Cover2_error := Cover2_opened AND Cover2_closed;
Cover3_error := Cover3_opened AND Cover3_closed;
// we are open, if all covers are open
isopen := cover3_opened AND cover2_opened;
// we are closed, if all covers are closed
isclosed := cover2_closed AND cover3_closed;
// error indicates an axis error on any axis
Cover2_timeout(IN := (open AND NOT Cover2_opened) OR (close AND NOT Cover2_closed), PT := T#30S);
Cover3_timeout(IN := (open AND NOT Cover3_opened) OR (close AND NOT Cover3_closed), PT := T#30S);

error_trigger(	SET1 := Cover2_error OR Cover2_timeout.Q OR Cover3_error OR Cover3_timeout.Q,
				RESET := reset,
				Q1 => Error);

Ready := NOT Error;

IF isopen THEN
	open := FALSE;
END_IF
IF isclosed THEN
	close := FALSE;
END_IF

Cover_status.0 := isopen;
Cover_status.1 := isclosed;
Cover_status.2 := Warning;
Cover_status.3 := Error;
Cover_status.4 := isopen;
Cover_status.5 := FALSE;
Cover_status.6 := Cover2_opened;
Cover_status.7 := Cover3_opened;
Cover_status.8 := FALSE;
Cover_status.9 := Cover2_closed;
Cover_status.10 := Cover3_closed;
Cover_status.11 := FALSE;
Cover_status.12 := Cover2_error;
Cover_status.13 := Cover3_error;

IF Cover_status <> LastStatus THEN
	LastStatus := Cover_status;
	MAIN.MQTTClient.Publish('telescope', 'cover', 'CoverIsOpen', BOOL_TO_STRING(isopen));
	MAIN.MQTTClient.Publish('telescope', 'cover', 'CoverIsClosed', BOOL_TO_STRING(isclosed));
	MAIN.MQTTClient.Publish('telescope', 'cover', 'CoverWarning', BOOL_TO_STRING(Warning));
	MAIN.MQTTClient.Publish('telescope', 'cover', 'CoverError', BOOL_TO_STRING(Error));
	MAIN.MQTTClient.Publish('telescope', 'cover', 'CoverStatus', WORD_TO_STRING(Cover_status));
END_IF

// A timeout occurs, when we open the cover, and the opened signal does not activate within n seconds.
// The same holds for closing the cover. This should not take longer then 10 seconds
Cover2_timeout(IN := NOT (Cover2_opened XOR Cover2_closed), PT := T#20S);
				
Cover3_timeout(IN := NOT (Cover3_opened XOR Cover3_closed), PT := T#20S);

Covers_Error_Event.OnMessage := 'Cover drive error';
IF Error THEN
	IF Cover3_error THEN 
		Covers_Error_Event.OnMessage := 'Cover 3 has a drive error.';
	END_IF
	IF Cover2_error THEN 
		Covers_Error_Event.OnMessage := 'Cover 2 has a drive error.';
	END_IF
END_IF


Covers_Error_event(	Trigger := Error, 
					Level := ADSLOG_MSGTYPE_ERROR);

Covers_Warning_event(	Trigger := Warning, 
						Level := ADSLOG_MSGTYPE_WARN);

// raise an error, if both opened and closed signals are activated
// handle RoboTel differently
Cover2_Event(Trigger := cover2_opened AND cover2_closed,
				Level := ADSLOG_MSGTYPE_ERROR, 
				OnMessage := 'Cover2: limit switch error');

Cover3_Event(Trigger := cover3_opened AND cover3_closed,
				Level := ADSLOG_MSGTYPE_ERROR, 
				OnMessage := 'Cover3: limit switch error');

//trigger an event, if we encounter a timeout
// handle RoboTel differently

Cover2_Timeout_Event(Trigger := Cover2_timeout.Q,
				Level := ADSLOG_MSGTYPE_ERROR, 
				OnMessage := 'Cover2: Timeout');

Cover3_Timeout_Event(Trigger := Cover3_timeout.Q,
				Level := ADSLOG_MSGTYPE_ERROR, 
				OnMessage := 'Cover3: Timeout');
// Log if we are opened
Covers_opened_event(Trigger := isopen,
					Level := ADSLOG_MSGTYPE_WARN,
					OnMessage := 'All covers are open');
//log if we are closed
Covers_closed_event(Trigger := isclosed,
					Level := ADSLOG_MSGTYPE_HINT,
					OnMessage := 'All covers are closed');

END_PROGRAM

// ---- POUs/NasmythControl.TcPOU
PROGRAM NasmythControl
VAR_INPUT
	// unlocks the brake and enables the drive
	enable:	BOOL;
	// resets the drive
	reset: BOOL;
	// turns the Nasmyth mirror to left port (seen from top)
	left:	BOOL;
	// turns the Nasmyth mirror to right port (seen from top)
	right:	BOOL;
END_VAR
VAR_OUTPUT
	// Nasmyth drive error
	error:	BOOL;
	// drive ready
	Ready:	BOOL;
	// Nasmyth points to right mirror
	Nasmyth_right:		BOOL;
	// Nasmyth points to left mirror
	Nasmyth_left:		BOOL;
END_VAR
VAR
	//move to derotator
	nasmyth_move_left	AT%Q*: BOOL;
	nasmyth_move_right	AT%Q*: BOOL;
	// delay for the Nasmyth holding brake
	Nasmyth_delay:		TON;
	// status word for MQTT message
	Nasmyth_status:		WORD;
	// last status word to trigger MQTT message if different
	LastStatus:			WORD;
	// unlock the holding brake
	Nasmyth_unlock:		BOOL;
	// holding brake is unlocked
	Nasmyth_unlocked:	BOOL;
	// event log of error
	NasmythEvent: 		FB_Eventlog;
	NasmythLeftEvent:	FB_Eventlog;
	NasmythRightEvent:	FB_Eventlog;
	Nasmyth_Timeout:	TON := (PT := T#10S);
END_VAR

// get the inputs
Nasmyth_left := GVL_Telescope.nasmyth_limit_right;
Nasmyth_right := GVL_Telescope.nasmyth_limit_left;

// disable command, if position has been reached or 
IF Nasmyth_left OR right THEN
	left := FALSE;
END_IF

IF  Nasmyth_right OR left THEN
	right := FALSE;
END_IF

Nasmyth_status.0 := Nasmyth_unlocked;
Nasmyth_status.1 := error;
Nasmyth_status.2 := Nasmyth_left;
Nasmyth_status.3 := Nasmyth_right;
Nasmyth_status.4 := Nasmyth_Timeout.Q;
Nasmyth_status.5 := Ready;

Nasmyth_unlock := enable AND (left OR right);
// report Nasmyth unlocked after n milliseconds										
Nasmyth_delay(
	IN := Nasmyth_unlock,
	PT := T#250MS,
	Q => Nasmyth_unlocked);

// set the outputs
GVL_Telescope.nasmyth_lock := Nasmyth_unlock;

Nasmyth_Timeout(IN := (left AND NOT Nasmyth_left) OR (right AND NOT Nasmyth_right));

IF Nasmyth_status <> LastStatus THEN
	LastStatus := Nasmyth_status;
	MAIN.MQTTClient.Publish('telescope', 'nasmyth', 'NasmythUnlocked', BOOL_TO_STRING(Nasmyth_unlocked));
	MAIN.MQTTClient.Publish('telescope', 'nasmyth', 'NasmythError', BOOL_TO_STRING(error));
	MAIN.MQTTClient.Publish('telescope', 'nasmyth', 'NasmythReady', BOOL_TO_STRING(Ready));
	MAIN.MQTTClient.Publish('telescope', 'nasmyth', 'NasmythIsLeft', BOOL_TO_STRING(Nasmyth_left));
	MAIN.MQTTClient.Publish('telescope', 'nasmyth', 'NasmythIsRight', BOOL_TO_STRING(Nasmyth_right));
END_IF


NasmythEvent(	Trigger := error, 
				Level := ADSLOG_MSGTYPE_ERROR,
				OnMessage := 'Nasmyth axis error',
				OffMessage := 'OK',
				OffLevel := ADSLOG_MSGTYPE_HINT);

NasmythLeftEvent(	Trigger := Nasmyth_left, 
					Level := ADSLOG_MSGTYPE_HINT,
					OnMessage := 'Nasmyth is on left port');

NasmythRightEvent(	Trigger := Nasmyth_right, 
					Level := ADSLOG_MSGTYPE_HINT,
					OnMessage := 'Nasmyth is on right port');

END_PROGRAM

// ---- POUs/FanControl.TcPOU
PROGRAM FanControl
VAR_INPUT
	// enable the fan controller
	enable: BOOL := TRUE;	
	// reset the fan controller
	reset :	BOOL;
END_VAR
VAR_OUTPUT
	// error condition
	error: BOOL;	
END_VAR
VAR
	// fan axis reference
	Fan_axis:		MDP5001_511_733_8E9CD54E;
	// measured temperature
	temperature:	REAL;
	// calculated velocity
	velocity:		INT;
	velocity_percentage:	REAL;
	lrVelocity:		LREAL;
	// issue temperature warning
	TemperatureWarning: FB_EventLog;
	MQTTTimer:		TON := (PT:=T#5S);
	sPayloadPub: STRING(255) := '';
	softreset:		BOOL;
END_VAR

(* Upper telescope cabinet fan control *)

// enable the fan as soon as main cabinet is ready AND temperature exceeds ambient temperature
Fan_axis.MDP5001_511_733_Output.MDP5001_733_Control_1.Enable := Transformer.power_OK AND NOT Reset AND (temperature > Environment.TemperatureDome);
// reset on MAIN reset
Fan_axis.MDP5001_511_733_Output.MDP5001_733_Control_1.Reset := reset OR softreset;
// calculate the temperatur from analog input
temperature := GVL_Telescope.temperature_cabinet / 100.0;

// set the fan velocity as a function of temperature difference
lrvelocity:= F_YREAL(temperature - Environment.TemperatureDome, 1.0, 2.0, 0, 32767) ;
velocity := LREAL_TO_INT(lrvelocity);

velocity_percentage := 100.0*INT_TO_REAL(velocity)/32767.0;
// apply the calculated velocity
Fan_axis.MDP5001_511_733_Output.MDP5001_733_Velocity := velocity;
// return the error condition
error := Fan_axis.MDP5001_511_733_Input.MDP5001_733_Status_1.Error;

MQTTTimer(IN:=TRUE);
IF MQTTTimer.Q THEN // publish new payload every second
	MQTTTimer(IN:=FALSE);
	sPayloadPub := 'electronics,location=dome,host=CX-4E6032,module=TelescopeCabinet ';
	MAIN.MQTTClient.Publish('electronics', 'dome', 'TelescopeCabinetTemperature', LREAL_TO_FMTSTR(Temperature, 2, TRUE));
	MAIN.MQTTClient.Publish('electronics', 'dome', 'FanVelocity', LREAL_TO_FMTSTR(velocity_percentage, 1, TRUE));
END_IF

TemperatureWarning(Trigger := temperature >= 40.0,
				Level := ADSLOG_MSGTYPE_WARN,
				FormatString := '%s',
				OnMessage := 'Telescope cabinet temperature exceeds 40 degrees Celsius');

END_PROGRAM

// ---- POUs/Transformer.TcPOU
PROGRAM Transformer
VAR
	// watchdog for trafo softstarter
	power_watchdog: 	TON;
	power_timer:		FB_timer;
	startup_timeout:	TIME := T#2S;
	power_error_state:	SR;
	// trafo failed to start after timeout
	power_failure:		BOOL;
	reset_error:		BOOL := FALSE;
	softstart_trafo:	BOOL;
	PowerEvent:			FB_EventLog;
	PowerLog:			FB_EventLog;
END_VAR

power_timer(bStart := GVL_Main.softstart_trafo, bStop := power_OK);
power_watchdog(IN := GVL_Main.softstart_trafo AND NOT power_OK,
				PT := startup_timeout,
				Q => power_failure);
power_error_state(SET1 := power_failure, RESET := reset_error);

GVL_Main.softstart_trafo := softstart_trafo AND NOT error;

PowerEvent(	
	Trigger := 		power_failure, 
	Level := 		ADSLOG_MSGTYPE_ERROR,
	FormatString :=	'%s',
	OnMessage := 	'Servo power FAILURE!',
	OffMEssage := 	'Servo power OK');
PowerLog(	
	Trigger := 		power_OK, 
	Level := 		ADSLOG_MSGTYPE_HINT,
	FormatString :=	'%s',
	OnMessage := 	'Mains power is ON',
	OffMEssage := 	'Mains power is OFF');

PROPERTY error : BOOL
GET
error := power_error_state.Q1;
END_GET
END_PROPERTY

PROPERTY power_ok : BOOL
// indicates the power state for the AX5000
GET
power_ok := GVL_main.power_available;
END_GET
END_PROPERTY

METHOD reset : BOOL
VAR_INPUT
END_VAR
IF error THEN
	reset_error := TRUE;
ELSE
	reset_error := FALSE;
END_IF
END_METHOD

METHOD start : BOOL
VAR_INPUT
END_VAR
softstart_trafo := TRUE;
END_METHOD

PROPERTY startup_time : TIME
GET
startup_time := power_timer.tDifference;
END_GET
SET
startup_timeout := startup_time;
END_SET
END_PROPERTY

METHOD stop : BOOL
VAR_INPUT
END_VAR
softstart_trafo := FALSE;
END_METHOD

END_PROGRAM

// ---- POUs/AuxiliaryControl.TcPOU
PROGRAM AuxiliaryControl
VAR
	// start delay for the dehumidifier to prevent overcurrent
	DeHumidifierOnDelay:	TON;
	DeHumidifierDelay: 		TON;
	DeHumidifier:			BOOL;
	pressure_voltage,
	pressure_Dewar,
	temperature_Dewar: 		REAL;
END_VAR
VAR CONSTANT
	humidity_high:			REAL := 75.0;
	humidity_low:			REAL := 65.0;
END_VAR

// turn off dehumidifier if dome is open
IF Environment.HumidityDome >= humidity_high AND DomeControl.DomeClosed THEN
	DeHumidifier := TRUE;
ELSIF Environment.HumidityDome < humidity_low OR DomeControl.DomeOpened OR Environment.Humidity < Environment.HumidityDome THEN
	DeHumidifier := FALSE;
END_IF
// start the dehumidifier, if we are above warning theshold for x hours
DeHumidifierDelay(IN := (Environment.HumidityDome > humidity_low) AND 
						(Environment.HumidityDome < humidity_high) AND
						DomeControl.DomeClosed,
					PT := T#6H);

// delay startup of the dehumidifier to prevent power-spike
DeHumidifierOnDelay(IN := DeHumidifier OR DeHumidifierDelay.Q, PT := T#5S, Q=> GVL_Dome.DeHumidifier);

pressure_voltage := F_YREAL(GVL_Auxiliary.pressure_Dewar, 0, 32767, 0.0, 10.0);
pressure_Dewar := LREAL_TO_REAL(EXPT(10.0, (1.5*pressure_voltage - 12.0)));
temperature_Dewar := GVL_Auxiliary.temperature_Dewar / 100.0;

IF Trigger(GVL_Dome.DeHumidifier) THEN
	MAIN.MQTTClient.Publish('dome', 'dome', 'WeatherBad', BOOL_TO_STRING(GVL_Dome.DeHumidifier));	
END_IF

END_PROGRAM

// ---- POUs/SafetyHandling.TcPOU
PROGRAM SafetyHandling
VAR
	restart_safety 	: TP;
	//safety_state 	: RS;
	start_delay 	: TON;
	ErrAck_Pulse	: TP;
	SafetyLog		: FB_EventLog;
END_VAR
VAR_OUTPUT
	Error			: BOOL;
END_VAR
VAR_INPUT
	remote_restart:		BOOL;
	remote_ErrAck:		BOOL;
	remote_run:			BOOL := TRUE;
END_VAR

// Safety can be stopped by pressing STOP and RESET on main panel
GVL_Safety.Run := MAIN.phase_available AND remote_run;
// power on delay for Safety RESTART after RUN=1
restart_safety(IN := MAIN.phase_available, PT := T#1S);
// RESTART Safety after pushing reset or power on delay
GVL_Safety.Restart := Main.reset OR restart_safety.Q OR remote_restart;

// wait n seconds after Start ...
start_delay(IN := MAIN.phase_available, PT := T#2S);
// ... and send ErrAck for n milliseconds
ErrAck_Pulse(IN := MAIN.phase_available AND start_delay.Q, PT := T#200MS);

// Error Acknowledgment: Turn key_switch OFF and press STOP 
GVL_Safety.ErrAck := (NOT GVL_Main.key_switch_remote)
					OR ErrAck_Pulse.Q OR remote_ErrAck;
					
Error := GVL_Safety.Error;

SafetyLog(Trigger := Error,
				Level := ADSLOG_MSGTYPE_ERROR,
				OnMessage := 'Safety Error! Emergency stop enganged!',
				OffMessage := 'Safety is OK.',
				OffLevel := ADSLOG_MSGTYPE_HINT);

END_PROGRAM

// ---- POUs/FunctionBlocks/FB_LightTimer.TcPOU
FUNCTION_BLOCK FB_LightTimer
VAR_INPUT
	IN: BOOL;
	PT: TIME := T#60S;
END_VAR
VAR_OUTPUT
	Q: BOOL;
END_VAR
VAR
	SR1 : SR;
	rtrig: R_TRIG;
	ton1 : TON;
END_VAR

(*
This is a simple light control based on a impulse switch.
The output Q goes high on the rising edge of the input IN.
The output Q stays high until the time PT runs out or another rising edge on IN is detected.
*)

// detect the rsing edge of the input
rtrig(CLK := IN);
// reset the input after PT time
ton1(IN := Q,
		PT := PT);
// sets the flip-flop on the first rising edge, reset it on the second rising edge or when time is up.
SR1(SET1 := rtrig.Q AND NOT Q,
	RESET := ton1.Q OR (Q AND rtrig.Q),
	Q1 => Q);

END_FUNCTION_BLOCK

// ---- POUs/FunctionBlocks/FB_MOONPOS.TcPOU
FUNCTION_BLOCK FB_MOONPOS
VAR_INPUT
	jd: LREAL;
END_VAR
VAR_OUTPUT
	ra, dec: LREAL;
	geolong, geolat, dis: LREAL;
END_VAR
VAR
	//npts: INT;
	//N_elements: INT;
	d: LREAL;
	//  form time in Julian centuries from 1900.0
	T: LREAL;
	// Mean longitude of the moon refered to mean equinox of the date in radians
	lprime: LREAL;
	// Mean longitude of the moon refered to mean equinox of the date in degrees
	lprimed: LREAL;
	// Sun's mean anomaly in radians
	M: LREAL;
	// Moons's mean anomaly in radians
	Mprime: LREAL;
	// Moon's argument of latitude
	F: LREAL;
	// Eccentricity of Earth's orbit around the Sun
	E ,E2: LREAL;
	// Additional arguments
	A1, A2, A3: LREAL;
	suml_add, sumb_add : LREAL;

	sinlng, coslng, sinlat, coslat: ARRAY [0..59] OF LREAL;
	ecorr1, ecorr2,ecorr3, ecorr4, i: INT;
	// argument for loop calculation
	arg : LREAL; 
	// longitude in radians 
	lambda : LREAL; 
	// latitude in radians
	beta : LREAL; 
	// true obliquity in degrees 
	epsilon: LREAL; 
	 // true obliquity in radians
	eps: LREAL;
	nlong, elong: LREAL;
	
	nutate:	FB_NUTATE;
END_VAR
VAR CONSTANT
	d_lng: ARRAY[0..59] OF INT := [0,2,2,0,0,0,2,2,2,2, 0,1,0,2,0,0,4,0,4,2, 2,1,1,2,2,4,2,0,2,2, 1,2,0,0,2,2,2,4,0,3, 2,4,0,2,2,2,4,0,4,1, 2,0,1,3,4,2,0,1,2,2];
	m_lng: ARRAY[0..59] OF INT := [0,0,0,0,1,0,0,-1,0,-1,1,0,1,0,0,0,0,0,0,1,1,0,1,-1,0,0,0,1,0,-1,0,-2,1,2,-2,0,0,-1,0,0,1,-1,2,2,1,-1,0,0,-1,0,1,0,1,0,0,-1,2,1,0,0];
    mp_lng: ARRAY[0..59] OF INT := [1,-1,0,2,0,0,-2,-1,1,0,-1,0,1,0,1,1,-1,3,-2,-1,0,-1,0,1,2,0,-3,-2,-1,-2,1,0,2,0,-1,1,0,-1,2,-1,1,-2,-1,-1,-2,0,1,4,0,-2,0,2,1,-2,-3,2,1,-1,3,-1];
	f_lng: ARRAY[0..59] OF INT := [0,0,0,0,0,2,0,0,0,0,0,0,0,-2,2,-2,0,0,0,0,0,0,0,0,0,0,0,0,2,0,0,0,0,0,0,-2,2,0,2,0,0,0,0,0,0,-2,0,0,0,0,-2,-2,0,0,0,0,0,0,0,-2];
	sin_lng: ARRAY[0..59] OF LREAL := [6288774,1274027,658314,213618,-185116,-114332,58793,57066,53322,
										 45758,-40923,-34720,-30383,15327,-12528,10980,10675,10034,8548,-7888,-6766,
 										-5163,4987,4036,3994,3861,3665,-2689,-2602,2390,-2348,2236,-2120,-2069,2048, 
 										-1773,-1595,1215,-1110,-892,-810,759,-713,-700,691,596,549,537,520,-487, 
 										 -399,-381,351,-340,330,327,-323,299,294,0.0];
	cos_lng: ARRAY[0..59] OF LREAL := [-20905355,-3699111,-2955968,-569925,48888,-3149,246158,-152138, 
  -170733,-204586,-129620,108743,104755,10321,0,79661,-34782,-23210,-21636, 
   24208,30824,-8379,-16675,-12831,-10445,-11650,14403,-7003,0,10056,6322, 
  -9884,5751,0,-4950,4130,0,-3958,0,3258,2616,-1897,-2117,2354,0,0,-1423, 
  -1117,-1571,-1739,0,-4421,0,0,0,0,1165,0,0,8752.0];
   d_lat: ARRAY[0..60] OF INT := [0,0,0,2,2,2,2,0,2,0,2,2,2,2,2,2,2,0,4,0,0,0,1,0,0,0,1,0,4,4,0,4,2,2,2,2,0,2,2,2,2,4,2,2,0,2,1,1,0,2,1,2,0,4,4,1,4,1,4,2];
   m_lat: ARRAY[0..60] OF INT := [0,0,0,0,0,0,0,0,0,0,-1,0,0,1,-1,-1,-1,1,0,1,0,1,0,1,1,1,0,0,0,0,0,0, 0,0,-1,0,0,0,0,1,1,0,-1,-2,0,1,1,1,1,1,0,-1,1,0,-1,0,0,0,-1,-2];
   mp_lat: ARRAY[0..60] OF INT := [0,1,1,0,-1,-1,0,2,1,2,0,-2,1,0,-1,0,-1,-1,-1,0,0,-1,0,1,1,0,0,3,0,-1,1,-2,0,2,1,-2,3,2,-3,-1,0,0,1,0,1,1,0,0,-2,-1,1,-2,2,-2,-1,1,1,-1,0,0];
   f_lat: ARRAY[0..60] OF INT :=[ 1,1,-1,-1,1,-1,1,1,-1,-1,-1,-1,1,-1,1,1,-1,-1,-1,1,3,1,1,1,-1,-1,-1,1,-1,1,-3,1,-3,-1,-1,1,-1,1,-1,1,1,1,1,-1,3,-1,-1,1,-1,-1,1,-1,1,-1,-1, -1,-1,-1,-1,1];
   sin_lat: ARRAY[0..60] OF LREAL := [5128122,280602,277693,173237,55413,46271,32573,17198,9266,8822, 8216,4324,4200,-3359,2463,2211,2065,-1870,1828,-1794,-1749,-1565,-1491, -1475,-1410,-1344,-1335,1107,1021,833,777,671,607,596,491,-451,439,422,  421,-366,-351,331,315,302,-283,-229,223,223,-220,-220,-185,181,-177,176,  166,-164,132,-119,115,107.0];

	coeff0: ARRAY [0..4] OF LREAL := [218.3164477, 481267.88123421, -0.0015786, 1.0/538841.0, -1.0/6.5194];
	coeff1: ARRAY [0..4] OF LREAL := [297.8501921, 445267.1114034, -0.0018819, 1.0/545868.0, -1.0/1.13065E8];
	coeff2: ARRAY [0..3] OF LREAL := [357.5291092, 35999.0502909, -0.0001536, 1.0/2.449E7, 0.0];
	coeff3: ARRAY [0..4] OF LREAL := [134.9633964, 477198.8675055, 0.0087414, 1.0/6.9699E4, -1.0/1.4712E7];
	coeff4: ARRAY [0..4] OF LREAL := [93.2720950, 483202.0175233, -0.0036539, -1.0/3.526, 1.0/8.6331];
	c: ARRAY [0..10] OF LREAL := [21.448,-4680.93,-1.55,1999.25,-51.38,-249.67,-39.05,7.12,27.87,5.79,2.45];
	dtor: LREAL := PI/180.0;
END_VAR



	t := (jd - 2451545.0)/36525.0;
 
	FOR i := 0 TO 4 DO
		lprimed := lprimed + coeff0[i]*EXPT(T, i);
		d := d + coeff1[i]*EXPT(T, i);
		M := M + coeff2[i]*EXPT(T, i);
		Mprime := Mprime + coeff3[i]*EXPT(T, i);
		F := F + coeff4[i]*EXPT(T, i);
	END_FOR
	lprimed := LMOD(lprimed, 360.0);
	Lprime := Lprimed * dtor;
	d := LMOD(d, 360.0) * dtor;
	M := LMOD(M, 360.0) * dtor; 
    Mprime := LMOD(Mprime, 2.0*PI) * dtor;
	F := LMOD(F, 360.0) * dtor;
    
    E := 1 - 0.002516*T - 7.4 - 6*T*T;
    E2 := E*E;

// Additional arguments
    A1 := (119.75 + 131.849*T) * dtor;
    A2 := (53.09 + 479264.290*T) * dtor;
    A3 := (313.45 + 481266.484*T) * dtor;
    suml_add := 3958*SIN(A1) + 1962*SIN(lprime - F) + 318*SIN(A2);
    sumb_add :=  -2235*SIN(lprime) + 382*SIN(A3) + 175*SIN(A1-F) +  175*SIN(A1 + F) + 127*SIN(Lprime - Mprime) -   115*SIN(Lprime + Mprime);

// Sum the periodic terms 

	geolong := lprimed + suml_add/1.0E6; 
	geolat := sumb_add/1.0E6; 
	dis := 385000.56;

	FOR i := 0 TO 59 DO
		// ecorr1 := where(ABS(m_lng) EQ 1);
		IF m_lng[i] = 1 THEN
			sinlng[i] := e*sin_lng[i];
			coslng[i] := e*cos_lng[i];
		END_IF
		// ecorr2 := where(ABS(m_lat) EQ 1);
		IF m_lat[i] = 1 THEN
			sinlat[ecorr2] := e*sin_lat[ecorr2];
		END_IF
	   // ecorr3 := where(ABS(m_lng) EQ 2);
		IF m_lng[i] = 2 THEN
			sinlng[i] := e2*sin_lng[i];
			coslng[i] := e2*cos_lng[i];
		END_IF
	   // ecorr4 := where(ABS(m_lat) EQ 2);
		IF m_lat[i] = 2 THEN
			sinlat[i] := e2*sin_lat[i];
		END_IF
		
		arg := d_lng[i]*d + m_lng[i]*m +mp_lng[i]*mprime + f_lng[i]*f;
		geolong := geolong + sinlng[i]*SIN(arg)/1.0E6;
	
		dis := dis + coslng[i]*COS(arg)/1.0E3;
	
		arg := d_lat[i]*d + m_lat[i]*m + mp_lat[i]*mprime + f_lat[i]*f;
		geolat := geolat + sinlat[i]*SIN(arg)/1.0E6;
		
	END_FOR

//Find the nutation in longitude
	nutate(jd := jd, nut_long => nlong, nut_obliq => elong);                     
	
	geolong := geolong + nlong/3.6E3;
	geolong := LMOD(geolong, 360.0);
	lambda := geolong*dtor;
	beta := geolat*dtor;

//Find mean obliquity and convert lambda,beta to RA, Dec
	epsilon := 23.433333333; // 23 deg 26 min 
	FOR i:=0 TO 10 DO
		epsilon := epsilon +  c[i]*EXPT(T/1.0E2, i)/3600.0;
	END_FOR
	
	eps := (epsilon + elong/3600.0 )*dtor;          //True obliquity in radians
	
	ra := ATAN2( SIN(lambda)*COS(eps) - TAN(beta)* SIN(eps), COS(lambda) );
	dec := ASIN( SIN(beta)*COS(eps) + COS(beta)*SIN(eps)*SIN(lambda) );

	ra := LMOD(ra/dtor, 360.0); 
	dec := dec/dtor;

END_FUNCTION_BLOCK

// ---- POUs/Functions/LREAL_TO_FMTESTR.TcPOU
FUNCTION LREAL_TO_FMTESTR : STRING
VAR_INPUT
	in         : LREAL; // 1.19412572985311e-6
    iPrecision : INT := 2;
    bRound     : BOOL := TRUE;
END_VAR
VAR
	lstring: STRING;
	ppos: INT;
	epos: INT;
	mantisse: LREAL;
	exponent: STRING;
END_VAR

lstring := LREAL_TO_STRING(in);
ppos := FIND(lstring, '.');
epos := FIND(lstring, 'e');
IF epos = 0 OR ppos = 0 THEN
	LREAL_TO_FMTESTR := LREAL_TO_FMTSTR(in, iPrecision, bRound);
	RETURN;
END_IF
mantisse := STRING_TO_LREAL(LEFT(lstring, epos-1)); // 1.19412572985311
exponent := RIGHT(lstring, LEN(lstring)-epos+1); // e-6
LREAL_TO_FMTESTR := CONCAT(LREAL_TO_FMTSTR(mantisse,iPrecision, bRound), exponent);

END_FUNCTION

// ---- GlobalTextList.TcGTLO
TEXTLIST GlobalTextList
  869 = 'brake open'
  518 = 'close brake'
  379 = 'Covers'
  462 = 'covers closed'
  683 = 'covers open'
  957 = 'Elevation enable'
  183 = 'go home'
  760 = 'goto'
  339 = 'Hydraulics'
  830 = 'Hydraulics start'
  664 = 'Hydraulics stop'
  157 = 'Hydraulik'
  101 = 'Licht'
  483 = 'Light'
  725 = 'open brake'
  470 = 'open cover'
  387 = 'park'
  252 = 'Poewr'
  597 = 'Power'
  182 = 'power'
  207 = 'pump running'
  596 = 'reset'
  851 = 'Reset'
  649 = 'start hydraulics'
  414 = 'stop hydraulics'
  661 = 'suction running'
  990 = 'Telescope control'
  422 = 'Text'
  39 = 'Track'
  34 = 'track'
END_TEXTLIST

// ---- VISUs/Visualization.TcVIS
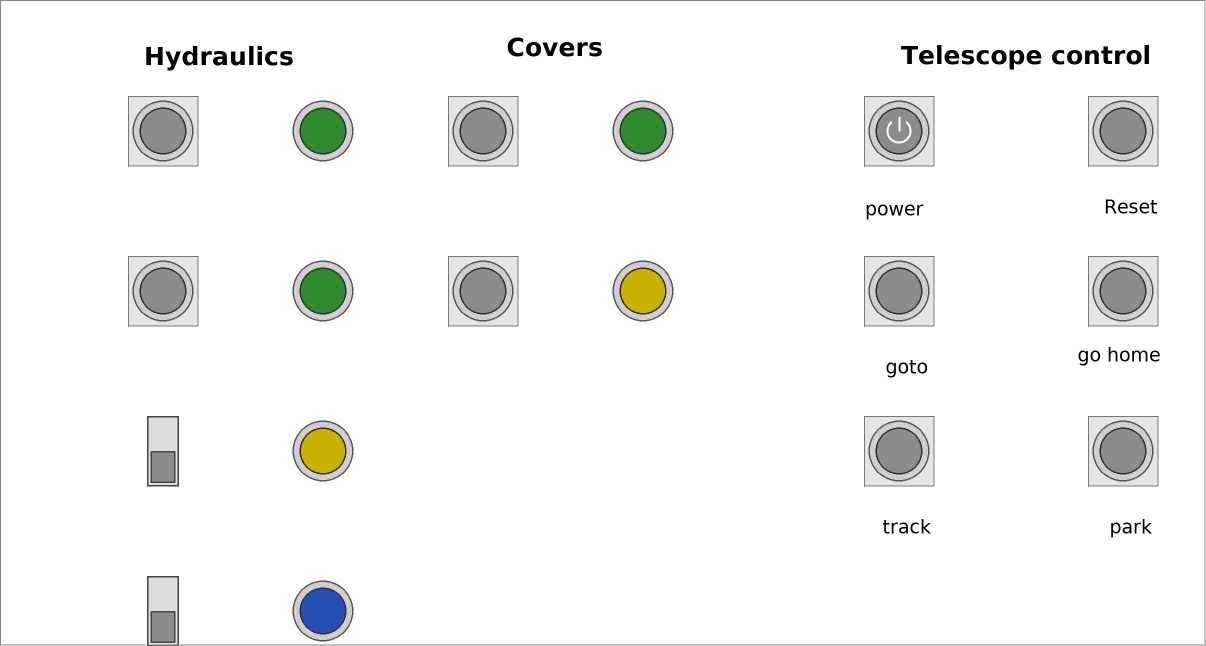
VISUALIZATION Visualization  // 1206x646
    PushSwitch (1088,96 70x70), tooltip "reset", variable: TelescopeControl.reset, behaviour: TAP, style: Switch-PushSwitch-Gray
    PushSwitch (1088,416 70x70), tooltip "park", variable: TelescopeControl.park, behaviour: TAP, style: Switch-PushSwitch-Gray
    Lamp1 (288,96 70x70), tooltip "pump running", variable: HydraulicsControl.pump_running, style: Lamp-Lamp1-Green
    Lamp1 (288,256 70x70), tooltip "suction running", variable: HydraulicsControl.suction_running, style: Lamp-Lamp1-Green
    PushSwitch (864,416 70x70), tooltip "Track", variable: TelescopeControl.track, behaviour: TAP, style: Switch-PushSwitch-Gray
    PowerSwitch (864,96 70x70), tooltip "Power", variable: TelescopeControl.power, behaviour: TOGGLE, style: Switch-PowerSwitch-Gray
    PushSwitch (1088,256 70x70), tooltip "go home", variable: TelescopeControl.gohome, behaviour: TAP, style: Switch-PushSwitch-Gray
    Lamp1 (288,416 70x70), tooltip "brake open", variable: HydraulicsControl.brake_open, style: Lamp-Lamp1-Yellow
    Label (800,192 189x34), "power"
    Label (1056,192 150x30), "Reset"
    Label (1056,512 150x30), "park"
    Label (1044,340 150x30), "go home"
    PushSwitch (864,256 70x70), tooltip "goto", variable: TelescopeControl.goto, behaviour: TAP, style: Switch-PushSwitch-Gray
    Label (832,512 150x30), "track"
    Label (832,352 150x30), "goto"
    Lamp1 (288,576 70x70), tooltip "Light", variable: GVL_Dome.Light, style: Lamp-Lamp1-Blue
    PushSwitch (128,96 70x70), tooltip "start hydraulics", variable: HydraulicsControl.start, behaviour: TOGGLE, style: Switch-PushSwitch-Gray
    PushSwitch (128,256 70x70), tooltip "stop hydraulics", variable: HydraulicsControl.stop, behaviour: TOGGLE, style: Switch-PushSwitch-Gray
    DipSwitch (128,576 70x70), tooltip "Licht", variable: MAIN.Lightbutton, behaviour: TOGGLE, style: Switch-DipSwitch-Gray
    DipSwitch (128,416 70x70), tooltip "open brake", variable: HydraulicsControl.open_brake, behaviour: TOGGLE, style: Switch-DipSwitch-Gray
    PushSwitch (448,96 70x70), tooltip "open cover", variable: CoverControl.open, behaviour: TOGGLE, style: Switch-PushSwitch-Gray
    PushSwitch (448,256 70x70), variable: CoverControl.close, behaviour: TOGGLE, style: Switch-PushSwitch-Gray
    Lamp1 (608,96 70x70), tooltip "covers open", variable: CoverControl.isopen, style: Lamp-Lamp1-Green
    Lamp1 (608,256 70x70), tooltip "covers closed", variable: CoverControl.isclosed, style: Lamp-Lamp1-Yellow
    Label (480,32 150x30), "Covers"
    Label (144,41 150x30), "Hydraulics"
    Label (899,40 254x30), "Telescope control"
END_VISUALIZATION
